TYPE ST_Recipe :
STRUCT
    stInfo           : ST_RecipeInfo;
    stSolventsTimes  : ST_RecipeSolventAndTimes;
    stVolumes        : ST_RecipeVolumes;
    stOtherParams    : ST_RecipeOtherParams;
END_STRUCT
END_TYPE

(* stored: Version 1.1.0.1, ProductVersion 3.1.4024.12
   DUT ST_Recipe: Id {f7b88f77-e2e0-4055-8c4a-415f0b4b34ca} *)
